TYPE IoChuckPsd :
STRUCT				
END_STRUCT
END_TYPE

(* stored: Version 1.1.0.1, ProductVersion 3.1.4024.12
   DUT IoChuckPsd: Id {32a741fb-190c-4e2f-b6f9-bf219c48c9b1} *)
